TYPE REAL_UNION :
UNION
    Value : REAL;
    Raw : UDINT;
END_UNION
END_TYPE

(* stored: Version 1.1.0.1
   DUT REAL_UNION: Id {45a8f752-e352-42e7-996a-402c3a7b3513} *)
